Staubli VAL3: Product.pjx

--- Product.pjx ---
Parameters version=s7.8.3 stackSize=5000 millimeterUnit=true
Program file=EditPath.pgx
Program file=getList.pgx
Program file=Init.pgx
Program file=InsertPath.pgx
Program file=Main.pgx
Program file=MainKey.pgx
Program file=OnF1.pgx
Program file=OnF2.pgx
Program file=OnF3.pgx
Program file=OnF4.pgx
Program file=OnF5.pgx
Program file=OnF6.pgx
Program file=OnF7.pgx
Program file=OnF8.pgx
Program file=readFileList.pgx
Program file=Refresh.pgx
Program file=RefreshList.pgx
Program file=Save.pgx
Program file=selectFile.pgx
Program file=selectPath.pgx
Program file=setPrd.pgx
Program file=start.pgx
Program file=stop.pgx
Data file=Product.dtx
Library alias=master path=Disk://template/normal/normal.pjx
Library alias=user path=Disk://userPage/USERPAGE.pjx
Library alias=PublicData path=Disk://PublicData/PublicData.pjx
Library alias=PublicProg path=Disk://PublicProg/PublicProg.pjx
Library alias=Path path=Disk://Path/Path.pjx
Library alias=Motion path=Disk://Motion/Motion.pjx
Library alias=SparePoint path=Disk://SparePoint/SparePoint.pjx

--- Product.dtx ---
bool bExit
bool bListRefresh
bool bUserRefresh
mdesc mNomSpeed
num nPage
num nSelected
public string sDeli[2]
  [0] = "A"
  [1] = "C"
public string sFileList
string sFolder = "Disk://Traj/"
string sItem = "paodpe"
string sList[2]
  [0] = "paodpe"
  [1] = "popo"
string sOutputFolder = "Disk://Traj/"
string sPathList
num nPrdIndex
string sNewPath
string sProductList
string sPrd

--- Main.pgx ---
program Main()
  local num l_nKey
begin
  //
  nPage=0
  do
    call Refresh()
    call RefreshList()
    call user:setList("产品",sList,bUserRefresh,bListRefresh,nSelected,sItem,l_nKey)
    bUserRefresh=false
    bListRefresh=false
    call MainKey(l_nKey)
    delay(0)
  until bExit

end

--- EditPath.pgx ---
program EditPath()
  local num l_nKey
begin
  //
  nPage=1
  bUserRefresh=bListRefresh=true
  do
    call Refresh()
    call RefreshList()
    call user:setList("路径",sList,bUserRefresh,bListRefresh,nSelected,sItem,l_nKey)
    bUserRefresh=false
    bListRefresh=false
    call MainKey(l_nKey)
    delay(0)
  until bExit
  nPage=0
  bUserRefresh=bListRefresh=true
  bExit=false
end

--- getList.pgx ---
program getList(string x_sPtPara, string& x_sOutPtpara[])
  local num l_nRes
  local num l_ni
begin
  //对参数x_sPtPara进行解析，得到相应信息

  call PublicProg:SplitChar(l_nRes,x_sPtPara,"/",x_sOutPtpara)

end

--- Init.pgx ---
program Init()
  local num l_ni
  local string l_sKey
begin
  //
  bUserRefresh=bListRefresh=true
  //
  bExit=false
  //
  call readFileList(sFolder,sFileList)
  //按照前缀sDeli选择相应的文件
  //call selectFile(sDeli,sFileList)
  //

  //call getList(PublicData:sPrd,sPrd)

  resize(sPrd,1,size(PublicData:sPrd))
  for l_ni=0 to size(PublicData:sPrd)-1
    sPrd[l_ni]=PublicData:sPrd[l_ni]
  endFor

  resize(sProductList,1,size(PublicData:sProductList))
  for l_ni=0 to size(PublicData:sProductList)-1
    sProductList[l_ni]=PublicData:sProductList[l_ni]
  endFor

end

--- InsertPath.pgx ---
program InsertPath()
  local string l_sProperty[3]
  local string l_sItem
begin
  l_sProperty[0]="轨迹"
  l_sProperty[1]="码垛盘"
  l_sProperty[2]="离散点"
  call user:SetProerty("",20,8,6,3,l_sProperty,l_sItem)

  if l_sItem==l_sProperty[0]
    //读取路径
    call readFileList(sFolder,sFileList)
    call selectFile(sDeli,sFileList)
    //
    call selectPath()
  elseIf l_sItem==l_sProperty[1]
    l_sProperty[0]="pallet1"
    l_sProperty[1]="pallet2"
    call user:SetProerty("",20,9,8,2,l_sProperty,l_sItem)
    if l_sItem!=""
      if sPathList[0]!="pallet1" and sPathList[0]!="pallet2"
        insert(sPathList[0])
        sPathList[0]=l_sItem
      else
        if sPathList[size(sPathList)-1]!="pallet1" and sPathList[size(sPathList)-1]!="pallet2"
          insert(sPathList[size(sPathList)])
          sPathList[size(sPathList)-1]=l_sItem
        else
          popUpMsg("码垛盘最多两个!")
        endIf
      endIf

    endIf
  else
    call SparePoint:setPoint("")
    call SparePoint:start()
    call SparePoint:getPoint(l_sItem)
    //popUpMsg(l_sItem)
    if l_sItem!=""
      if sPathList[nSelected]!=""
        nSelected=nSelected+1
        insert(sPathList[nSelected])
        sPathList[nSelected]=l_sItem
      else
        sPathList[nSelected]=l_sItem
      endIf

    endIf
    endIf

  //
end

--- MainKey.pgx ---
program MainKey(num x_nKey)
  local num l_nKey
begin
  //
  switch x_nKey
    //编辑
    case 271,270
      call OnF1()
    break
    //取反
    case 272
      call OnF2()
    break
    //删除
    case 273
      call OnF3()
    break
    //模拟
    case 274
      call OnF4()
    break
    //
    case 275
    break
    //
    case 276
      call OnF6()
    break
    //save
    case 277
      call OnF7()
    break
    //返回
    case 278,255
      call OnF8("是否返回")
    break
  endSwitch
end

--- OnF1.pgx ---
program OnF1()
  local bool l_bRes
begin
  //
  switch nPage
    case 0
      if sItem!=""
        nPrdIndex=nSelected
        call getList(sProductList[nSelected],sPathList)
        call EditPath()
      else
       popUpMsg("空路径不能编辑")
      endIf

    break
    case 1
      if sItem!=""
        call Path:EditMain(sItem)
      else
        popUpMsg("空路径不能编辑")
      endIf

    break
    //
    case 2
      sNewPath=sItem
      popUpMsg("新增加路径："+sItem)
    break
  endSwitch
  bUserRefresh=bListRefresh=true
end

--- OnF2.pgx ---
program OnF2()
  local num l_ni
  local bool l_bRes
  local string l_sItem
begin
  //
  switch nPage
    //新建产品
    case 0
      call setPrd(sList,l_sItem)
      if l_sItem!=""
        if sPrd[nSelected]!=""
          nSelected=nSelected+1
          insert(sPrd[nSelected])
          insert(sProductList[nSelected])
        endIf
        sPrd[nSelected]=l_sItem
        sProductList[nSelected]=""
      endIf
    break
    //插入路径
    case 1
      call InsertPath()
    break
  endSwitch
  bUserRefresh=bListRefresh=true
end

--- OnF3.pgx ---
program OnF3()
  local string l_sYesNo[2]
  local num l_i
begin

  //
  if sList[nSelected]!=""
    l_sYesNo[0]="是"
    l_sYesNo[1]="否"
    call user:questionDialog("是否删除?",l_sYesNo,l_i)
    if l_i==0 or l_i==1
      switch nPage
        case 0
          if size(sPrd)==1
            sPrd[nSelected]=""
            sProductList[nSelected]=""
          else
            delete(sPrd[nSelected])
            delete(sProductList[nSelected])
            if nSelected>=1
              nSelected=nSelected-1
            endIf
          endIf

        break
        case 1
          if size(sList)==1
            sList[nSelected]=""
          else
            delete(sList[nSelected])
            if nSelected>=1
              nSelected=nSelected-1
            endIf

          endIf
        break
      endSwitch
      bListRefresh=true
    else
      popUpMsg("没有可以删除的项目")
    endIf
  endIf
  bUserRefresh=true
end

--- OnF4.pgx ---
program OnF4()
begin
  //
  PublicData:bSimulaiton=true
  call Motion:AllMotion(sItem)
  bUserRefresh=true
end

--- OnF6.pgx ---
program OnF6()
  local string l_sProperty[2]
  local string l_sItem
begin
  switch nPage
    case 0
      l_sProperty[0]="设置"
      l_sProperty[1]="取消"
      call user:SetProerty("",26,9,6,2,l_sProperty,l_sItem)
      if l_sItem==l_sProperty[0]
        if sItem==""
          popUpMsg("没有产品")
        else
          PublicData:sStartPrd=sItem
          PublicData:libSave()
          popUpMsg("选择产品"+sItem+"为自启动")

        endIf
      else
        PublicData:sStartPrd=""
        PublicData:libSave()
        popUpMsg("自启动取消")
      endIf
      bUserRefresh=bListRefresh=true
    break
    case 1
    break
  endSwitch
end

--- OnF7.pgx ---
program OnF7()
begin
  //
  call Save()
end

--- Refresh.pgx ---
program Refresh()
begin
  //
  if bUserRefresh
    cls()
    userPage()
    switch nPage
      case 0
        gotoxy(1,1)
        put("F1->编辑")
        gotoxy(1,13)
        put("F1")
        gotoxy(1,2)
        put("F2->新建")
        gotoxy(6,13)
        put("F2")
        gotoxy(1,3)
        put("F3->删除")
        gotoxy(11,13)
        put("F3")
        gotoxy(1,4)
        put("F4->模拟")
        gotoxy(16,13)
        put("F4")
        //
        gotoxy(1,6)
        put("F6->设置/取消自启动")
        gotoxy(26,13)
        put("F6")
        gotoxy(1,7)
        put("F7->保存")
        gotoxy(31,13)
        put("F7")
        gotoxy(1,8)
        put("F8->返回")
        gotoxy(36,13)
        put("F8")
      break
      case 1
        gotoxy(1,1)
        put("F1->编辑")
        gotoxy(1,13)
        put("F1")
        gotoxy(1,2)
        put("F2->插入")
        gotoxy(6,13)
        put("F2")
        gotoxy(1,3)
        put("F3->删除")
        gotoxy(11,13)
        put("F3")
        //        gotoxy(1,4)
        //        put("F4->模拟")
        //        gotoxy(16,13)
        //        put("F4")
        //
        //    gotoxy(1,6)
        //    put("F6->")
        //    gotoxy(26,13)
        //    put("")
        gotoxy(1,7)
        put("F7->保存")
        gotoxy(31,13)
        put("F7")

        gotoxy(1,8)
        put("F8->返回")
        gotoxy(36,13)
        put("F8")
      break
      case 2
        gotoxy(1,1)
        put("F1->确定")
        gotoxy(1,13)
        put("F1")
        gotoxy(1,2)
        //        put("F2->插入")
        //        gotoxy(6,13)
        //        put("F2")
        //        gotoxy(1,3)
        //        put("F3->删除")
        //        gotoxy(11,13)
        //        put("F3")
        //        //        gotoxy(1,4)
        //        //        put("F4->模拟")
        //        //        gotoxy(16,13)
        //        //        put("F4")
        //        //
        //        //    gotoxy(1,6)
        //        //    put("F6->")
        //        //    gotoxy(26,13)
        //        //    put("")
        //        gotoxy(1,7)
        //        put("F7->保存")
        //        gotoxy(31,13)
        //        put("F7")

        gotoxy(1,8)
        put("F8->返回")
        gotoxy(36,13)
        put("F8")
      break
    endSwitch

  endIf
end

--- RefreshList.pgx ---
program RefreshList()
  local num l_ni
begin
  //
  switch nPage
    case 0
      if bListRefresh
        resize(sList,1,size(sPrd))
        for l_ni=0 to size(sList)-1
          sList[l_ni]=sPrd[l_ni]
        endFor
      endIf
    break
    case 1
      resize(sList,1,size(sPathList))
      for l_ni=0 to size(sList)-1
        sList[l_ni]=sPathList[l_ni]
      endFor
    break
    //
    case 2
      resize(sList,1,size(sFileList))
        for l_ni=0 to size(sList)-1
          sList[l_ni]=sFileList[l_ni]
        endFor
    break
  endSwitch
end

--- Save.pgx ---
program Save()
  local num l_ni
begin

  switch nPage
    //产品
    case 0
      resize(PublicData:sPrd,1,size(sPrd))
      for l_ni=0 to size(sPrd)-1
        PublicData:sPrd[l_ni]=sPrd[l_ni]
      endFor
      //
      resize(PublicData:sProductList,1,size(sProductList))
      for l_ni=0 to size(sList)-1
        PublicData:sProductList[l_ni]=sProductList[l_ni]
      endFor
      PublicData:libSave()
      popUpMsg("保存成功!")
    break
    //每一个产品里的路径
    case 1
      //产品保存
      resize(PublicData:sPrd,1,size(sPrd))
      for l_ni=0 to size(sPrd)-1
        PublicData:sPrd[l_ni]=sPrd[l_ni]
      endFor
      //
      resize(PublicData:sProductList,1,size(sProductList))
      sProductList[nPrdIndex]=sList[0]
      for l_ni=1 to size(sList)-1
        sProductList[nPrdIndex]=sProductList[nPrdIndex]+"/"+sList[l_ni]
      endFor
      PublicData:sProductList[nPrdIndex]=sProductList[nPrdIndex]
      PublicData:libSave()
      popUpMsg("保存成功!")
    break
  endSwitch
end

--- selectFile.pgx ---
public program selectFile(string& x_sDelimiter[], string& x_sList[])
  local num l_ni
  local num l_nj
begin
  //
  for l_nj=0 to size(x_sList)-1
    if x_sList[l_nj]!=""
      for l_ni=0 to size(x_sDelimiter)-1
        if left(x_sList[l_nj],1)==x_sDelimiter[l_ni]
          l_ni=size(x_sDelimiter)
        endIf
        if l_ni==size(x_sDelimiter)-1
          delete(x_sList[l_nj])
          l_nj=l_nj-1
        endIf
      endFor
    endIf

  endFor
end

--- selectPath.pgx ---
program selectPath()
  local num l_nKey
  local num l_nSelected
begin
  //
  nPage=2
  bUserRefresh=bListRefresh=true
  sNewPath=""
  l_nSelected=nSelected
  do
    call Refresh()
    call RefreshList()
    call user:setList("路径",sList,bUserRefresh,bListRefresh,nSelected,sItem,l_nKey)
    bUserRefresh=false
    bListRefresh=false
    call MainKey(l_nKey)
    delay(0)
  until bExit
  //
  if sPathList[l_nSelected]!=""
    if sNewPath!=""
      insert(sPathList[l_nSelected+1])
      sPathList[l_nSelected+1]=sNewPath
    endIf
  else
    sPathList[l_nSelected]=sNewPath
  endIf

  nPage=1
  bUserRefresh=bListRefresh=true
  bExit=false
end

--- setPrd.pgx ---
program setPrd(string& x_sInOut[], string& x_sOut)
  local string l_sItemName
begin
  //
  x_sOut=""
  call PublicProg:addListItem(l_sItemName,x_sInOut,"P")
  if l_sItemName!=""
    //建立
    if x_sInOut[0]!=""
      insert(x_sInOut[size(x_sInOut)])
    endIf
    x_sInOut[size(x_sInOut)-1]=l_sItemName
    x_sOut=l_sItemName
    call user:listadd(l_sItemName)
  endIf
end
